// TIA Portal V17 export
// export: Created 2025-08-05T09:35:58.7290248Z, ExportSetting WithDefaults, DisplayName Totally Integrated Automation Portal, DisplayVersion V17, DisplayName TIA Portal Openness, DisplayVersion V17, DisplayName TIA Portal Version Control Interface, DisplayVersion V17, DisplayName SINAMICS Startdrive Advanced, DisplayVersion V17, DisplayName SINAMICS Startdrive G130, G150, S120, S150, SINAMICS MV, S210, DisplayVersion V17, DisplayName SINAMICS Startdrive G110M, G120, G120C, G120D, G120P, G115D, DisplayVersion V17, DisplayName STEP 7 Professional, DisplayVersion V17, DisplayName STEP 7 Safety, DisplayVersion V17, DisplayName WinCC Advanced, DisplayVersion V17
DATA_BLOCK "Call_DB"   // DB7
VERSION : 0.1
// stored: AutoNumber true, DBAccessibleFromOPCUA true, DBAccessibleFromWebserver true, InstanceOfName Call, InstanceOfType FB
"Call"
   // VAR
   //    LaserComm_API_Instance { S7_SetPoint := 'True'} : Array[0..1] of "LaserComm_API";
   //    Dummy_Cereal_Number { S7_SetPoint := 'True'} : Array[1..32] of Char;
   //    Dummy_Part_Type { S7_SetPoint := 'True'} : Array[1..18] of Char;
   // END_VAR
BEGIN
END_DATA_BLOCK
